(* Schneider Machine Expert - Basic project ProyekFillingBottle, file version 2.5.0.0 *)
(* ProjectInformations: Name=New project *)

HARDWARE
  Cpu 0: TM221CE24T
  EthernetConfiguration: NetworkName=M221, IpAllocationMode=FixedAddress, IpAddress=0.0.0.0, SubnetMask=0.0.0.0
  SerialLineConfiguration: Baud=Baud19200, Parity=ParityEven, DataBits=DataBits8, StopBits=StopBits1, PhysicalMedium=PhysicalMediumRs485, TransmissionMode=TransmissionModeModbusRtu, SlaveId=1, Addressing=SlaveAddressing
  MastTask: UsePeriodScanMode=false, PeriodScan=100
  FastTask: Period=255
  CpuBehavior: StartingMode=StartAsPreviousState, AutoSaveRamOnEeprom=true, WatchdogPeriod=250

SYMBOLS  (address, symbol, comment, settings)
  %TM0        [Preset=3, Base=OneSecond]
  %C0         [Preset=999]
  %I0.2     SENSOR

POU New POU
  (* SectionNumber=1 *)

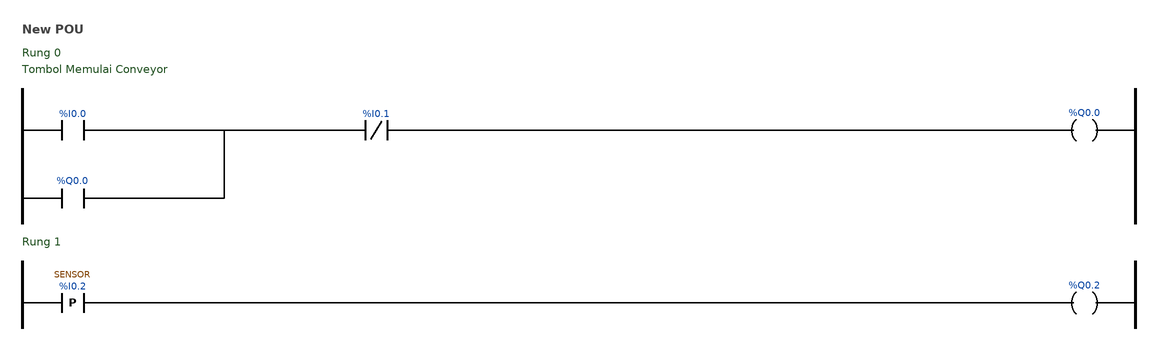

// Rung 0
// Tombol Memulai Conveyor
  LD %I0.0
  OR %Q0.0
  ANDN %I0.1
  ST %Q0.0
  // as ST:
  //   %Q0.0 := (%I0.0 OR %Q0.0) AND NOT %I0.1;

// Rung 1
  LDR %I0.2               (* SENSOR *)
  ST %Q0.2
  // as ST:
  //   %Q0.2 := RISING(SENSOR);

POU New POU
  (* SectionNumber=2 *)

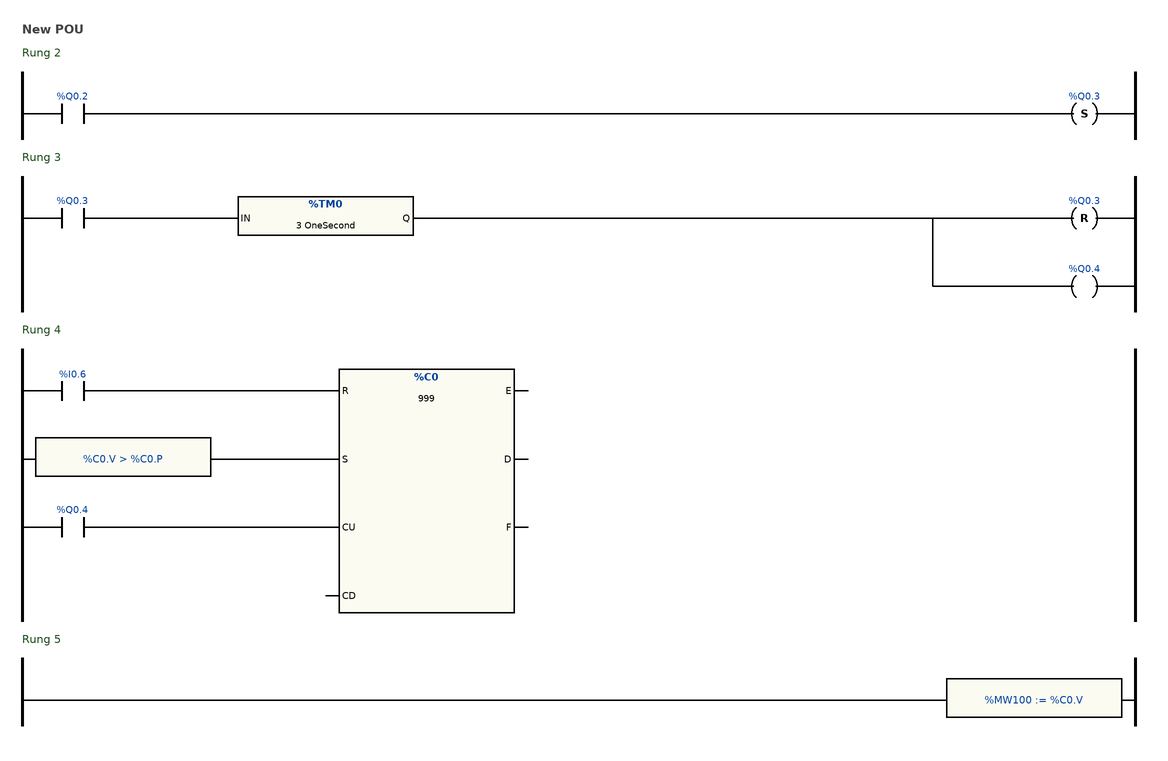

// Rung 2
  LD %Q0.2
  S %Q0.3
  // as ST:
  //   IF %Q0.2 THEN %Q0.3 := TRUE; END_IF;

// Rung 3
  BLK %TM0
  LD %Q0.3
  IN
  OUT_BLK
  LD Q
  R %Q0.3
  ST %Q0.4
  END_BLK
  // as ST:
  //   %TM0(IN := %Q0.3);
  //   IF %TM0.Q THEN %Q0.3 := FALSE; END_IF;
  //   %Q0.4 := %TM0.Q;

// Rung 4
  BLK %C0
  LD %I0.6
  R
  LD [ %C0.V > %C0.P ]
  S
  LD %Q0.4
  CU
  END_BLK
  // as ST:
  //   %C0(R := %I0.6, S := %C0.V > %C0.P, CU := %Q0.4);

// Rung 5
  LD 1
  [ %MW100 := %C0.V ]
  // as ST:
  //   %MW100 := %C0.V;
